// TIA Portal V18 export
DATA_BLOCK "Sys"   // DB3000
{ S7_Optimized_Access := 'FALSE' }
VERSION : 0.1
// stored: AutoNumber false, DBAccessibleFromOPCUA true, DBAccessibleFromWebserver true, IsOnlyStoredInLoadMemory false, IsWriteProtectedInAS false
   VAR RETAIN
      COM : Struct   // Common
         AlwaysOFF : Bool := FALSE;
         AlwaysON : Bool := TRUE;
         FlashTime100mS : Bool := TRUE;   // Hardware Clock Memory 0.1S
         FlashTime200mS : Bool := TRUE;   // Hardware Clock Memory 0.2S
         FlashTime500mS : Bool := FALSE;   // Hardware Clock Memory 0.5S
         FlashTime1S : Bool := FALSE;   // Hardware Clock Memory 1S
         FlashTime2S : Bool := TRUE;   // Hardware Clock Memory 2S
         SpareBit : Bool := FALSE;
         PLCRestarted : Bool := TRUE;
      END_STRUCT;
      SpareB1 : Array[0..7] of Byte;
      DateTime : Struct   // DBX10.0
         Set : Date_And_Time := DT#1990-01-01-00:00:00;
         Read : Date_And_Time := DT#2025-03-12-08:03:05.785;
         Trigger : Bool := FALSE;   // Set
         ReturnValueRead : Int := 0;
         ReturnValueSet : Int := 0;
      END_STRUCT;
      SpareB2 : Array[0..17] of Byte;
      ScanTime : Struct   // DBX50.0
         CyclePrevious : Int := 14;
         CycleMax : Int := 23;
         CycleMin : Int := 9;
      END_STRUCT;
      RETVALI : Int := 0;
      RETVALW : Word := 16#0000;
      VersionManagement : Struct
         ProductLineName : String := 'Assembly Line';
         ProjectNumber : String[20] := 'SZ23055';
         "PLC IP Addr" : Array[0..3] of UInt;
         "HMI IP Addr" : Array[0..3] of UInt;
         PLCVersion : Array[0..1] of UInt;
         HMIVersion : Array[0..1] of UInt;
         "TIA Version" : String := 'TIA V18';
         StationID : Int := 10;
         HMIPageID : Int := 0;
      END_STRUCT;
   END_VAR
BEGIN
   SpareB1[0..7] := 16#00;
   SpareB2[0..17] := 16#00;
   VersionManagement."PLC IP Addr"[0] := 192;
   VersionManagement."PLC IP Addr"[1] := 168;
   VersionManagement."PLC IP Addr"[2..3] := 10;
   VersionManagement."HMI IP Addr"[0] := 192;
   VersionManagement."HMI IP Addr"[1] := 168;
   VersionManagement."HMI IP Addr"[2] := 45;
   VersionManagement."HMI IP Addr"[3] := 11;
   VersionManagement.PLCVersion[0] := 1;
   VersionManagement.PLCVersion[1] := 0;
   VersionManagement.HMIVersion[0] := 1;
   VersionManagement.HMIVersion[1] := 0;
END_DATA_BLOCK
